{attribute 'GeneratedUsingTerminal: EL3403-0000-0017'}
{attribute addProperty BoxType "EL3403-0000-0017"}
{attribute addProperty Id "Missing_zero_crossing_AAT %I*BOOL1Missing_zero_crossing_BAT %I*BOOL1Missing_zero_crossing_CAT %I*BOOL1Phase_sequence_errorAT %I*BOOL1Sync_ErrorAT %I*BOOL1"}
{attribute addProperty CRC "265319072"}
{attribute addProperty Size "5"}
TYPE PM_Status_data_0FD072A0 :
STRUCT
	{attribute addProperty Name "Missing_zero_crossing_A"}
	Missing_zero_crossing_A AT %I* : BOOL;
	{attribute addProperty Name "Missing_zero_crossing_B"}
	Missing_zero_crossing_B AT %I* : BOOL;
	{attribute addProperty Name "Missing_zero_crossing_C"}
	Missing_zero_crossing_C AT %I* : BOOL;
	{attribute addProperty Name "Phase_sequence_error"}
	Phase_sequence_error AT %I* : BOOL;
	{attribute addProperty Name "Sync_Error"}
	Sync_Error AT %I* : BOOL;
END_STRUCT
END_TYPE

(* stored: Version 1.2.0.0, ProductVersion 3.1.4024.9
   DUT PM_Status_data_0FD072A0: Id {ff41a593-40b3-49e7-bd03-05dafbe7f082} *)
